(* PLC project Generated.project, CODESYS CODESYS V3.5 SP19 Patch 1 *)
(* stored: creationDateTime 2026-08-29T23:00:21.513526, modificationDateTime 2026-08-29T23:00:21.513526 *)

(* ═══════════════════════════════════════════════════════════════ 🎚️ ST_fbModes_Autorisations — Bus d'autorisations du mode machine ─────────────────────────────────────────────────────────────── 📄 Doc métier : DOC/AF/AF_Partie-05_Modes_Maintenance_v2.1.md DOC/AF/AF_Partie-02_Architecture_Programme_v3.2.md §2 🎯 Produit par FB_Modes (via PRG_03_Modes_Cycle) Consommé par : Cycle, Safety, Treuils, Translation, Supervision, Acquisition 🎯 Producteur unique : FB_Modes (via PRG_03_Modes_Cycle) ═══════════════════════════════════════════════════════════════ *)
TYPE ST_fbModes_Autorisations : STRUCT
  Mode : E_Mode;  (* Mode arbitré (DISABLE/N1/N2/SEMI_AUTO) *)
  SyncEnable : BOOL;  (* Synchro M1/M2 (logique positive) *)
  InhibitM1 : BOOL;  (* Inhibition M1 (MAINT_N2 only) *)
  InhibitM2 : BOOL;  (* Inhibition M2 (MAINT_N2 only) *)
  JoystickWinchSelectArbitrated : INT;  (* 0=M1+M2 couplés nominal, 1=M1, 2=M2 (unitaires MAINT_N2) *)
  HomingApproachEnable : BOOL;  (* Dépassement butée haut (N2) *)
  MaintenanceM3TargetEnable : BOOL;  (* Cible Translation Maintenance (N2 only) *)
  ModeChangePendingBlocked : BOOL;  (* AF-05 §4bis — matrice de maintenance ⚠️ Ces trois champs sont des FAITS/DIAGS publiés, pas des autorisations : ils restent vrais même quand le FB est neutralisé par Enable=FALSE (état persistant à remonter à l'IHM). 🚦 Demande de changement de mode REFUSÉE : les treuils *)
  HomingRequiredM1 : BOOL;  (* ne sont pas à l'arrêt mécanique confirmé (contacteurs retombés ET frein serré ET |v| < seuil). Le mode courant est maintenu. IHM : « arrêter les treuils avant de changer de mode ». 🧭 M1 : re-homing obligatoire avant tout retour SEMI_AUTO *)
  HomingRequiredM2 : BOOL;  (* (usage effectif d'un override/bypass position en maintenance) 🧭 M2 : idem *)
END_STRUCT;
END_TYPE

(* values of E_Mode: DISABLE: Mode Désactivé / Veille de sécurité (sorties bloquées); MAINT_N1: Manuel Niveau 1 : Pilotage unitaire avec toutes sécurités actives; MAINT_N2: Manuel Niveau 2 : Pilotage dégradé (droits étendus + bypasses autorisés); SEMI_AUTO: Mode Semi-Automatique (séquenceur automatique) *)

{attribute 'qualified_only'}
{attribute 'strict'}
TYPE E_Mode : (DISABLE := 0, MAINT_N1 := 1, MAINT_N2 := 2, SEMI_AUTO := 3);
END_TYPE
